FUNCTION_BLOCK FB_Module EXTENDS FB_Component
VAR_INPUT
END_VAR
VAR_OUTPUT
END_VAR
VAR
	fbLogger:					FB_LoggerFactory;
	fbTcLogger:					FB_TcLogger;
	fbAlarm:					FB_Alarm;
END_VAR

METHOD PUBLIC M_Attach
VAR_INPUT
	Component:		I_Component;
END_VAR
Component.P_Event.P_Logger:= fbLogger;
Component.P_Observer.M_Attach(THIS^);
fbObserver.M_Attach(Component);
END_METHOD

METHOD PUBLIC M_Cycle
VAR_INPUT
END_VAR
fbAlarm.M_Cycle();
SUPER^.M_Cycle();
END_METHOD

METHOD PUBLIC M_Dettach
VAR_INPUT
	Component:		I_Component;
END_VAR
Component.P_Event.P_Logger:= 0;
Component.P_Observer.M_Detach(THIS^);
fbObserver.M_Detach(Component);
END_METHOD

METHOD PROTECTED M_Initialise : BOOL
VAR_INPUT
END_VAR
M_Initialise:= SUPER^.M_Initialise();

fbEvent.P_Logger:= fbLogger;
fbLogger.M_Add(fbAlarm);
fbLogger.M_Add(fbTcLogger);
END_METHOD

METHOD PROTECTED M_Resetting : BOOL
VAR_INPUT
END_VAR
VAR
	nIndex:					DINT;
END_VAR
fbAlarm.M_Reset();

M_Resetting:= TRUE;
WHILE nIndex < fbObserver.nLength DO
	fbObserver.M_Index(nIndex).M_Request(E_Request.Reset);
	nIndex:= nIndex +1;
END_WHILE
END_METHOD

METHOD PROTECTED M_Running
VAR_INPUT
END_VAR
END_METHOD

METHOD PROTECTED M_Starting : BOOL
VAR_INPUT
END_VAR
VAR
	nIndex:					DINT;
END_VAR
M_Starting:= TRUE;
WHILE nIndex < fbObserver.nLength DO
	M_Starting:= M_Starting AND fbObserver.M_Index(nIndex).M_Request(E_Request.Start);
	nIndex:= nIndex +1;
END_WHILE
END_METHOD

END_FUNCTION_BLOCK

(* stored: Version 1.1.0.1
   POU FB_Module: Id {0d3fc497-598e-0d21-1617-ce19be6391a0}, SpecialFunc None
   Method M_Attach: Id {579d130b-ed70-0843-1869-7cfcfab74d3d}
   Method M_Cycle: Id {ed9a21fb-3ec5-0016-04de-0d3b7ca7722a}
   Method M_Dettach: Id {a667402b-5023-09c1-34b6-30ca3f961f61}
   Method M_Initialise: Id {d2ecc479-1ed6-0218-1db6-cf2c288ac295}
   Method M_Resetting: Id {a610a2e6-39fb-0abb-32e8-2f742935aded}
   Method M_Running: Id {8879f60a-43a4-0568-363b-e25a42eddf0c}
   Method M_Starting: Id {5a9fb78b-3ed4-0195-387d-72e3c96a0cbd} *)
